KUKA KRL data list: main.dat

&ACCESS RVP
&REL 5
&COMMENT Main Program Data
DEFDAT main
  ; --- Local Point Declarations for Go-to-Definition & Diff ---
  DECL E6POS P1={X 1200.5, Y -450.0, Z 950.0, A 0.0, B 90.0, C 0.0, S 2, T 35}
  DECL E6POS P2={X 1200.5, Y -450.0, Z 800.0, A 0.0, B 90.0, C 0.0, S 2, T 35}
  DECL E6POS PICK_POINT={X 1450.0, Y 300.0, Z 650.0, A 45.0, B 0.0, C 180.0, S 6, T 19}
  DECL E6POS PLACE_POINT={X 1800.0, Y -200.0, Z 500.0, A -90.0, B 0.0, C 180.0, S 6, T 19}

  ; --- Local Motion Parameters ---
  DECL FDAT F1={TOOL_NO 1, BASE_NO 1, IPO_FRAME #BASE}
  DECL FDAT F2={TOOL_NO 1, BASE_NO 1, IPO_FRAME #BASE}
  DECL LDAT LPDAT1={VEL 2.0, ACC 100.0, APO_DIST 100.0, APO_FAC 50.0, AXIS_VEL 100.0, AXIS_ACC 100.0}
  DECL PDAT PPDAT1={VEL 100.0, ACC 100.0, APO_DIST 50.0}
ENDDAT
